(* PLC project Tc2_Utilities.FB_GetRouterStatusInfo Demo, tc3-libraries-kb TwinCAT 3.1 *)
(* stored: creationDateTime 2026-05-11T00:00:00, modificationDateTime 2026-05-11T00:00:00 *)

PROGRAM P_Demo_FB_GetRouterStatusInfo
  VAR
    fbFB_GetRouterStatusInfo : FB_GetRouterStatusInfo;  (* FB_GetRouterStatusInfo 实例 *)
    bRead : BOOL := FALSE;
    stRouterInfo : ST_AmsRouterStatusInfo;
    bBusy_ : BOOL;
    bErrFlag : BOOL;
    nErrCode : UDINT;
  END_VAR

// =============================================================================
// 场景：HMI 网络诊断页每秒读 Router 状态。
// 价值：路由器级观测，比 ping 精确。
// 验证：触发后观察 stRouterInfo.nMessages 在变；正常工况 nLostMessages 应为 0。
// 验证步骤：
//   1. 右键 PLC 项目 → Import PLCopenXML → 选本文件
//   2. 引用 Tc2_Utilities（References → Add library）
//   3. 编译 → 登录 → 运行；按上方『验证』行的指示在线写值观察
// =============================================================================

fbFB_GetRouterStatusInfo(
    bExecute := bRead,
    tTimeout := DEFAULT_ADS_TIMEOUT,
    stStatusInfo => stRouterInfo,
    bBusy => bBusy_,
    bErr => bErrFlag,
    nErrId => nErrCode
);
END_PROGRAM
